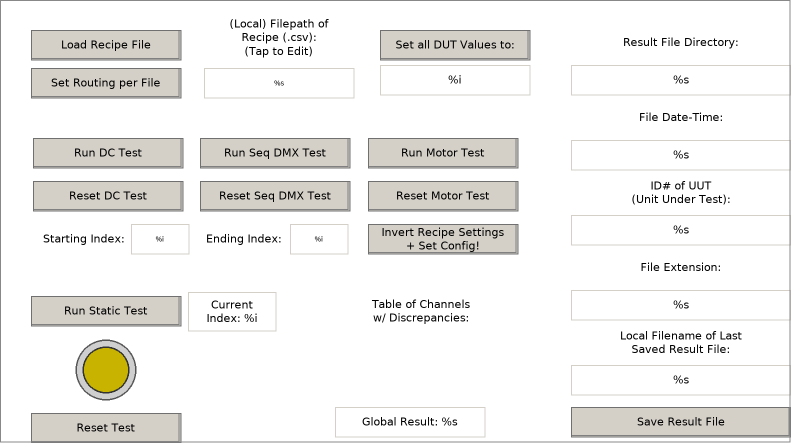
VISUALIZATION Visualization  // 791x443
    Button (31,30 150x30), "Load Recipe File", invisible if: DMXTest.iParseFile<>0
        tap P_TextModeRead.r_tFileChg.CLK
    Label (204,9 150x57), "(Local) Filepath of Recipe (.csv): (Tap to Edit)"
    Textfield (204,68 150x30), "%s", text variable: P_TextModeRead.sFilePathHMI
        OnMouseClick: write the text variable via Edit
    Textfield (335,407 150x30), "Global Result: %s"
    Label (356,296 130x30), "Table of Channels w/ Discrepancies:"
    Label (571,177 220x31), "ID# of UUT (Unit Under Test):"
    Textfield (571,215 220x30), "%s", text variable: P_TextModeWrite.sDUTIDNr
        OnMouseClick: write the text variable via VisuDialogs.Keypad
    Button (571,407 220x30), "Save Result File"
        tap P_TextModeWrite.r_tSaveResultFile.CLK
    Label (571,327 220x31), "Local Filename of Last Saved Result File:"
    Textfield (571,365 220x30), "%s", text variable: P_TextModeWrite.sFileName
    Label (571,102 220x31), "File Date-Time:"
    Textfield (571,140 220x30), "%s", text variable: P_TextModeWrite.sTimestamp
        tap P_TextModeWrite.r_tUpdateTimestamp.CLK p3779583253=TRUE
    Label (571,27 220x31), "Result File Directory:"
    Label (571,252 220x31), "File Extension:"
    Textfield (571,290 220x30), "%s", text variable: P_TextModeWrite.sFileExtension
        OnMouseClick: write the text variable via VisuDialogs.Keypad
    Textfield (571,65 220x30), "%s", text variable: P_TextModeWrite.sFileDir
        OnMouseClick: write the text variable via VisuDialogs.Keypad
    Lamp1 (71,335 70x70), variable: DMXTest.xDMXSeqTestInProgressOnce, style: Lamp-Lamp1-Yellow
    Button (31,296 150x30), "Run Static Test"
        tap DMXTest.rt_RunStaticTest.CLK
    Button (31,413 150x30), "Reset Test", invisible if: DMXTest.iCompareStaticSM<>120
        tap DMXTest.rt_ResetTest.CLK p3779583253=TRUE
    Button (31,68 150x30), "Set Routing per File", invisible if: DMXTest.iSetConfig<>0
        tap DMXTest.r_tSetConfig.CLK
    Textfield (188,292 88x39), "Current Index: %i", text variable: DMXTest.uiLoopRcvIndex
    Button (380,30 150x30), "Set all DUT Values to:"
        tap DMXTest.r_tSetDUTVal.CLK
    Textfield (380,65 150x30), "%i", text variable: DMXTest.usiDUTVal
        OnMouseClick: write the text variable via InputWithLimits, min 0, max 255
    Button (200,138 150x30), "Run Seq DMX Test"
        tap DMXTest.rt_RunSeqTestOnce.CLK p3779583253=TRUE
    Button (200,181 150x30), "Reset Seq DMX Test"
        tap DMXTest.rt_ResetTestSeq.CLK p3779583253=TRUE
    Button (33,138 150x30), "Run DC Test"
        tap DMXTest.rt_RunSeqTestOnceDC.CLK p3779583253=TRUE
    Button (33,181 150x30), "Reset DC Test"
        tap DMXTest.rt_ResetTestSeqDC.CLK p3779583253=TRUE
    Button (368,138 150x30), "Run Motor Test"
    Button (368,181 150x30), "Reset Motor Test"
    Textfield (131,224 58x30), "%i", text variable: DMXTest.uiStartingIndex
        OnMouseClick: write the text variable via Edit
    Textfield (290,224 58x30), "%i", text variable: DMXTest.uiEndingIndex
        OnMouseClick: write the text variable via Edit
    Label (44,225 80x28), "Starting Index:"
    Label (204,225 80x28), "Ending Index:"
    Button (368,224 150x30), "Invert Recipe Settings + Set Config!"
        tap DMXTest.R_TInvertRecipe.CLK p3779583253=TRUE
END_VISUALIZATION

(* stored: Version 1.1.0.1, ProductVersion 3.1.4024.9
   Visu Visualization: Id {1a37950b-72f8-448c-a809-243b1f3c3855} *)
